// TIA Portal V18 export
VAR_GLOBAL   // PLC tag table "Default tag table"
   System_Byte AT %MB1 : Byte;
   FirstScan AT %M1.0 : Bool;
   DiagStatusUpdate AT %M1.1 : Bool;
   AlwaysTRUE AT %M1.2 : Bool;
   AlwaysFALSE AT %M1.3 : Bool;
   Clock_Byte AT %MB0 : Byte;
   Clock_10Hz AT %M0.0 : Bool;
   Clock_5Hz AT %M0.1 : Bool;
   "Clock_2.5Hz" AT %M0.2 : Bool;
   Clock_2Hz AT %M0.3 : Bool;
   "Clock_1.25Hz" AT %M0.4 : Bool;
   Clock_1Hz AT %M0.5 : Bool;
   "Clock_0.625Hz" AT %M0.6 : Bool;
   "Clock_0.5Hz" AT %M0.7 : Bool;
   "!!tagName:Contactor1_FeedbackInput$$" AT %I0.1 : Bool;
   "!!tagName:Contactor1_Output$$" AT %Q0.1 : Bool;
   "!!tagName:Contactor1_QBadInput$$" AT %I10.1 : Bool;
   "!!tagName:Contactor2_FeedbackInput$$" AT %I0.2 : Bool;
   "!!tagName:Contactor3_FeedbackInput$$" AT %I0.3 : Bool;
   "!!tagName:Contactor4_FeedbackInput$$" AT %I0.4 : Bool;
   "!!tagName:Contactor2_Output$$" AT %Q0.2 : Bool;
   "!!tagName:Contactor2_QBadInput$$" AT %I10.2 : Bool;
   "!!ITERATOR_STRINGS$$" AT %I0.5 : Bool;
   "!!tagName:EncoderSensor1$$" AT %I20.1 : Bool;
   "!!tagName:EncoderSensor2$$" AT %I20.2 : Bool;
   "!!tagName:SorterRunningIOC$$" AT %I20.6 : Bool;
   "!!tagName:DoorClosedCh1$$" AT %I30.1 : Bool;
   "!!tagName:DoorClosedCh2$$" AT %I30.2 : Bool;
   "!!tagName:DoorClosedDiagInput$$" AT %I30.0 : Bool;
   "!!tagName:DoorOpenRequest$$" AT %I140.6 : Bool;
   "!!tagName:DoorReset$$" AT %I140.7 : Bool;
   "!!tagName:DoorResetLamp$$" AT %Q140.7 : Bool;
   "!!tagName:DoorSolenoidUnlock$$" AT %Q140.6 : Bool;
   "!!tagName:GlobalEmergencyReset$$" AT %I50.0 : Bool;
END_VAR
